// TIA Portal V16 export
// export: Created 2023-03-29T11:03:36.0209651Z, ExportSetting WithDefaults, DisplayName Totally Integrated Automation Portal, DisplayVersion V16 Update 6, DisplayName TIA Portal Version Control Interface, DisplayVersion V16 Update 2, DisplayName TIA Portal Openness, DisplayVersion V16 Update 6, DisplayName STEP 7 Professional, DisplayVersion V16 Update 6, DisplayName STEP 7 Safety, DisplayVersion V16, DisplayName WinCC Advanced, DisplayVersion V16 Update 6
DATA_BLOCK "ERR_ErrorBufferFull"   // DB106
{ S7_Optimized_Access := 'TRUE' }
VERSION : 0.1
// stored: AutoNumber false, DBAccessibleFromOPCUA true, IsOnlyStoredInLoadMemory false, IsRetainMemResEnabled false, IsWriteProtectedInAS false, MemoryReserve 0
   VAR
      Error { S7_SetPoint := 'True'} : ErrorStruct;
   END_VAR
   VAR RETAIN
      SoftwareError { S7_SetPoint := 'True'} : Array[0..4] of "stt_ERR_SoftwareError";
      GetError { S7_SetPoint := 'True'} : Array[0..27] of "stt_ERR_GetError";
      CounterDiagStatusUpdate : UInt;
   END_VAR
BEGIN
END_DATA_BLOCK
